(* IEC 61131-3 sources: xpxp/gpt-5, 22 files *)

(* ---- 11.st ---- *)
FUNCTION Sign : INT
VAR_INPUT
    x : REAL;
END_VAR
IF x > 0.0 THEN
    Sign := 1;
ELSIF x < 0.0 THEN
    Sign := -1;
ELSE
    Sign := 0;
END_IF;
RETURN;
END_FUNCTION

(* ---- 14.st ---- *)
FUNCTION FC1001 : BOOL
VAR_INPUT
	MEW: REAL; // Measured value
	SP: REAL;  // Switching value (setpoint)
	HYS: REAL; // Hysteresis in percent of |SP|
END_VAR
VAR_IN_OUT
 	OUT:BOOL;  // Latched output state
END_VAR
VAR
 	P_HYS: REAL; // Absolute hysteresis value derived from percent
END_VAR

// Calculate absolute hysteresis; ensure non-negative percentage
IF HYS < 0.0 THEN
	P_HYS := 0.0;
ELSE
	P_HYS := ABS(SP) * HYS * 0.01;
END_IF

// Hysteresis behavior:
// - Turn ON when measured value exceeds SP
// - Turn OFF when measured value falls below SP - P_HYS
// - Otherwise, retain previous state to avoid fluttering
IF MEW > SP THEN
	OUT := TRUE;
ELSIF MEW < (SP - P_HYS) THEN
	OUT := FALSE;
END_IF

// Function result mirrors the output state
FC1001 := OUT;
RETURN;

(* ---- 15.st ---- *)
FUNCTION FC1002 : BOOL
VAR_INPUT
	E_A, SENSOR: BOOL;
	ZEITW: TIME;
END_VAR
VAR_IN_OUT
	ZEIT:TON;
	P_HU, P_AL: BOOL;
END_VAR

(* Drive timer based on system enable and sensor *)
ZEIT(IN := (E_A AND SENSOR), PT := ZEITW);

(* Alarm latch logic *)
IF NOT E_A THEN
	P_AL := FALSE;
ELSE
	IF P_AL THEN
		P_AL := TRUE; (* keep latched until system is turned off *)
	ELSIF ZEIT.Q THEN
		P_AL := TRUE; (* latch alarm after sustained detection *)
	ELSE
		P_AL := FALSE;
	END_IF
END_IF

(* Horn logic: active only during early detection window *)
IF E_A THEN
	IF SENSOR AND NOT P_AL THEN
		P_HU := TRUE;
	ELSE
		P_HU := FALSE;
	END_IF
ELSE
	P_HU := FALSE;
END_IF

(* Function return indicates system ON status *)
FC1002 := E_A;

(* ---- 18.st ---- *)
FUNCTION FC1003 : VOID
VAR_INPUT
    IN_R:REAL;
    IN_MAX, IN_MIN:REAL;
    OUT_MAX, OUT_MIN:REAL;
END_VAR
VAR_OUTPUT
    OUT_R:REAL;
    FEH:BOOL;
END_VAR
VAR_TEMP
    DIFF1, DIFF2:REAL;
END_VAR

(* Initialize error flag *)
FEH := FALSE;

(* Calculate input and output spans *)
DIFF1 := IN_MAX - IN_MIN;
DIFF2 := OUT_MAX - OUT_MIN;

(* Validate input span to avoid division by zero *)
IF ABS(DIFF1) <= 1.0e-30 THEN
    FEH := TRUE;
    OUT_R := OUT_MIN; (* Safe fallback output *)
    RETURN;
END_IF

(* Normalize input to 0..1 with saturation *)
OUT_R := (IN_R - IN_MIN) / DIFF1;
IF OUT_R < 0.0 THEN
    OUT_R := 0.0;
ELSIF OUT_R > 1.0 THEN
    OUT_R := 1.0;
END_IF

(* Scale to output range *)
OUT_R := OUT_MIN + OUT_R * DIFF2;

END_FUNCTION

(* ---- 1.st ---- *)
FUNCTION_BLOCK FB_AlarmManager
VAR
	xAllOn : BOOL;
	xAllOff : BOOL;

	xAlarm1 : BOOL;
    xAlarm2 : BOOL;
END_VAR

IF xAllOff THEN
	xAlarm1 := FALSE;
	xAlarm2 := FALSE;
	xAllOff := FALSE;
	xAllOn := FALSE;
ELSIF xAllOn THEN
	xAlarm1 := TRUE;
	xAlarm2 := TRUE;
	xAllOn := FALSE;
END_IF

END_FUNCTION_BLOCK

(* ---- 10.st ---- *)
FUNCTION_BLOCK FB_Sigmoid
VAR_INPUT
    X : REAL;
END_VAR
VAR_OUTPUT
    Y : REAL;
END_VAR
VAR
    z : LREAL;    // Intermediate exponential value
    t : LREAL;    // Temporary result in LREAL for precision
END_VAR

// Numerically stable sigmoid implementation:
// if x >= 0: sigmoid(x) = 1 / (1 + exp(-x))
// else:       sigmoid(x) = exp(x) / (1 + exp(x))
IF X >= 0.0 THEN
    z := EXP(LREAL(-X));
    t := 1.0 / (1.0 + z);
    Y := REAL(t);
ELSE
    z := EXP(LREAL(X));
    t := z / (1.0 + z);
    Y := REAL(t);
END_IF
END_FUNCTION_BLOCK

(* ---- 12.st ---- *)
FUNCTION_BLOCK FB_Sinh
VAR
    X : REAL;
END_VAR

(* Compute hyperbolic sine of X in-place using the exponential function.
   Includes simple saturation and piecewise evaluation to mitigate overflow. *)

(* Soft-limit X to a safe computational range for REAL to reduce overflow risk *)
X := LIMIT(-88.0, X, 88.0);

IF X > 80.0 THEN
    (* For large positive X, sinh(X) ≈ 0.5 * exp(X) *)
    X := 0.5 * EXP(X);
ELSIF X < -80.0 THEN
    (* For large negative X, sinh(X) ≈ -0.5 * exp(-X) *)
    X := -0.5 * EXP(-X);
ELSE
    (* General case: sinh(X) = (e^X - e^-X) / 2 *)
    X := 0.5 * (EXP(X) - EXP(-X));
END_IF

END_FUNCTION_BLOCK

(* ---- 13.st ---- *)
FUNCTION_BLOCK FB_FindNumberWithAbort
VAR CONSTANT
    MAXNUMBERS : UINT := 99;
END_VAR
VAR
    aNumbers : ARRAY[0..MAXNUMBERS] OF INT; // Input list of numbers (0..99)
    nCnt : INT;                             // Index/result: 0..99 if found; 100 if not found
END_VAR

// Initialize index
nCnt := 0;

// Search through the list with two abort conditions:
// 1) EXIT when number 10 is found.
// 2) Terminate when end of list is reached (nCnt > MAXNUMBERS).
REPEAT
    IF aNumbers[nCnt] = 10 THEN
        EXIT;
    END_IF
    nCnt := nCnt + 1;
UNTIL nCnt > INT(MAXNUMBERS) END_REPEAT;

(* ---- 16.st ---- *)
FUNCTION_BLOCK FB_TrafficLight
VAR
    North_green : BOOL;
    North_yellow : BOOL;
    North_red : BOOL;
    East_green : BOOL;
    East_yellow : BOOL;
    East_red : BOOL;
    T1 : TON;
END_VAR

(* Free-running 10s cycle using TON *)
T1(IN := NOT T1.Q, PT := T#10s);

(* Default all off *)
North_green := FALSE;
North_yellow := FALSE;
North_red := FALSE;
East_green := FALSE;
East_yellow := FALSE;
East_red := FALSE;

(* Phase selection based on elapsed time *)
IF (T1.ET < T#5s) THEN
    (* 0ms - 5000ms *)
    North_green := TRUE;
    East_red := TRUE;
ELSIF (T1.ET < T#5500ms) THEN
    (* 5000ms - 5500ms *)
    North_yellow := TRUE;
    East_red := TRUE;
ELSIF (T1.ET < T#9500ms) THEN
    (* 5500ms - 9500ms *)
    North_red := TRUE;
    East_green := TRUE;
ELSE
    (* 9500ms - 10000ms *)
    North_red := TRUE;
    East_yellow := TRUE;
END_IF;

END_FUNCTION_BLOCK

(* ---- 17.st ---- *)
FUNCTION_BLOCK FB_WeatherStation
VAR
    aiOutside : INT;       // Outside temperature [°C], read from analog input
    aiHumidity: INT;       // Relative humidity [%]
    sShowText : STRING[80];// Display text for house
END_VAR

// Temperature classification with nested humidity evaluation
IF aiOutside < 18 THEN
    // Below comfort temperature
    sShowText := 'Cold';
ELSIF aiOutside > 25 THEN
    // Above comfort temperature
    sShowText := 'Hot';
ELSE
    // Temperature within 18..25°C: evaluate humidity
    IF (aiHumidity >= 40) AND (aiHumidity <= 75) THEN
        sShowText := 'Opt';
    ELSE
        sShowText := 'Temp. OK';
    END_IF
END_IF

(* ---- 19.st ---- *)
FUNCTION_BLOCK FB1005
VAR_INPUT
    START:BOOL;
    DICKE, V_MAX, V_MIN:REAL;
END_VAR
VAR_OUTPUT
    D_MAX, D_MIN:REAL;
    P1:BOOL;
END_VAR
VAR
    FO:BOOL;
END_VAR

(* Rising edge detection of START: initialize new measurement cycle *)
IF (START AND NOT FO) THEN
    (* Initialize min/max with first sample of the new cycle *)
    D_MAX := DICKE;
    D_MIN := DICKE;
END_IF

(* While measuring, continuously update min/max *)
IF START THEN
    IF DICKE > D_MAX THEN
        D_MAX := DICKE;
    END_IF
    IF DICKE < D_MIN THEN
        D_MIN := DICKE;
    END_IF
END_IF

(* Evaluate reject light based on tolerance band.
   Safety: If V_MIN > V_MAX (invalid band), force reject. *)
IF V_MIN <= V_MAX THEN
    P1 := (D_MIN < V_MIN) OR (D_MAX > V_MAX);
ELSE
    P1 := TRUE;
END_IF

(* Store previous START state for edge detection *)
FO := START
END_FUNCTION_BLOCK

(* ---- 2.st ---- *)
FUNCTION_BLOCK FB_BinomialCoefficient
VAR_INPUT
    N : INT;
    K : INT;
    i : INT;
END_VAR
VAR_OUTPUT
    C : ULINT;
    Valid : BOOL;
    Error : BOOL;
    ErrorID : UINT;
END_VAR
VAR
    nEff : UDINT;
    kEff : UDINT;
    j : UDINT;
    res : ULINT;
    numTerm : ULINT;
    denTerm : ULINT;
    gcd : ULINT;
    temp : ULINT;
    rem : ULINT;
END_VAR

(* Default outputs *)
Error := FALSE;
Valid := FALSE;
ErrorID := UINT#0;
C := ULINT#0;

(* Validate inputs *)
IF (N < 0) OR (K < 0) THEN
    Error := TRUE;
    ErrorID := UINT#10; (* Negative inputs not allowed *)
    RETURN;
END_IF

IF K > N THEN
    Error := TRUE;
    ErrorID := UINT#11; (* K must be <= N *)
    RETURN;
END_IF

(* Prepare effective parameters and use symmetry k = min(K, N-K) *)
nEff := UDINT(N);
kEff := UDINT(K);
IF kEff > (nEff - kEff) THEN
    kEff := nEff - kEff;
END_IF

res := ULINT#1;

(* Trivial cases *)
IF kEff = UDINT#0 THEN
    C := res; (* C(N,0) = 1 *)
    Valid := TRUE;
    RETURN;
END_IF

(* Multiplicative method with GCD reduction to control growth:
   res = product_{j=1..k} (n-k+j)/j
*)
FOR j := UDINT#1 TO kEff DO
    numTerm := ULINT(nEff - kEff + j);  (* numerator term *)
    denTerm := ULINT(j);                 (* denominator term *)

    (* Reduce (res, denTerm) by their GCD *)
    gcd := res;
    temp := denTerm;
    WHILE temp <> ULINT#0 DO
        rem := gcd MOD temp;
        gcd := temp;
        temp := rem;
    END_WHILE
    IF gcd > ULINT#1 THEN
        res := res / gcd;
        denTerm := denTerm / gcd;
    END_IF

    (* Reduce (numTerm, denTerm) by their GCD *)
    gcd := numTerm;
    temp := denTerm;
    WHILE temp <> ULINT#0 DO
        rem := gcd MOD temp;
        gcd := temp;
        temp := rem;
    END_WHILE
    IF gcd > ULINT#1 THEN
        numTerm := numTerm / gcd;
        denTerm := denTerm / gcd;
    END_IF

    (* Apply the reduced multiply/divide step *)
    res := res * numTerm;
    res := res / denTerm;
END_FOR

C := res;
Valid := TRUE
END_FUNCTION_BLOCK

(* ---- 20.st ---- *)
FUNCTION_BLOCK INTERLOCK
VAR_INPUT
    I1 : BOOL;
    I2 : BOOL;
    TL : TIME;
END_VAR
VAR_OUTPUT
    Q1 : BOOL;
    Q2 : BOOL;
END_VAR
VAR
    T1 : TOF;
    T2 : TOF;
END_VAR

(* Clamp the dead time to a minimum of 0 ms *)
IF TL < T#0ms THEN
    T1.PT := T#0ms;
    T2.PT := T#0ms;
ELSE
    T1.PT := TL;
    T2.PT := TL;
END_IF;

(* Timers monitor the opposite output to enforce dead time after switch-off *)
T1.IN := Q2; (* Blocks Q1 while Q2 is TRUE or has been TRUE within TL *)
T2.IN := Q1; (* Blocks Q2 while Q1 is TRUE or has been TRUE within TL *)

(* Execute timers *)
T1();
T2();

(* Interlock logic with deterministic priority to Q1 when both are eligible *)
IF (I1 AND NOT T1.Q) THEN
    Q1 := TRUE;
    Q2 := FALSE;
ELSIF (I2 AND NOT T2.Q) THEN
    Q1 := FALSE;
    Q2 := TRUE;
ELSE
    Q1 := FALSE;
    Q2 := FALSE;
END_IF;

(* ---- 21.st ---- *)
FUNCTION_BLOCK BURNER
VAR_INPUT
    IN : BOOL;
    STAGE2 : BOOL;
    OVER_TEMP : BOOL;
    OIL_TEMP : BOOL := TRUE;
    FLAME : BOOL;
    RST : BOOL;
    RST_TIMER : BOOL;
    PRE_HEAT_TIME : TIME := t#5s;
    PRE_VENT_TIME : TIME := t#15s;
    PRE_IGNITE_TIME : TIME := t#15s;
    POST_IGNITE_TIME : TIME := t#25s;
    STAGE2_DELAY : TIME := t#10s;
    SAFETY_TIME : TIME := t#5s;
    LOCKOUT_TIME : TIME := t#10s;
    MULTIPLE_IGNITION : BOOL := TRUE;
    KW1 : REAL;
    KW2 : REAL;
END_VAR
VAR_OUTPUT
    MOTOR : BOOL;
    COIL1 : BOOL;
    COIL2 : BOOL;
    PRE_HEAT : BOOL;
    IGNITE : BOOL;
    FAIL : BOOL;
    KWH : REAL;
    STATUS : BYTE;
END_VAR
VAR_IN_OUT
    RUNTIME1 : UDINT;
    RUNTIME2 : UDINT;
    CYCLES : UDINT;
END_VAR
VAR
    state : INT;
    last : TIME;
    tx : TIME;
    last_change : TIME;
    timer1 : TON;
    timer2 : TON;
    oil_temp_last : BOOL; (* used as last RST state for rising edge detection *)
    cycles2 : UDINT;      (* snapshot of RUNTIME1 at Stage1 start, used for Stage2 delay *)
END_VAR

(* Initialize to Standby on first scan *)
IF state = 0 THEN
    state := 110; (* Standby *)
    FAIL := FALSE;
    STATUS := 110;
END_IF

(* Reset runtime and energy counters on request *)
IF RST_TIMER THEN
    RUNTIME1 := 0;
    RUNTIME2 := 0;
    CYCLES := 0;
    KWH := 0.0;
    cycles2 := 0;
END_IF

(* Default outputs off; will be enabled per state below *)
MOTOR := FALSE;
COIL1 := FALSE;
COIL2 := FALSE;
PRE_HEAT := FALSE;
IGNITE := FALSE;

(* Over-temperature immediate lockout *)
IF OVER_TEMP AND NOT FAIL THEN
    FAIL := TRUE;
    STATUS := 9; (* boiler overheating contact has tripped *)
    state := 1000; (* Lockout state *)
    (* Prepare lockout timer1 *)
    timer1.IN := TRUE;
    timer1.PT := LOCKOUT_TIME;
END_IF

(* Lockout handling *)
IF state = 1000 THEN
    (* Ensure all actuators are off during lockout *)
    MOTOR := FALSE;
    COIL1 := FALSE;
    COIL2 := FALSE;
    PRE_HEAT := FALSE;
    IGNITE := FALSE;

    (* Run lockout timer *)
    timer1.PT := LOCKOUT_TIME;
    timer1.IN := NOT timer1.Q; (* keep running until elapsed *)

    (* Require RST low during lockout and accept rising edge after timer elapsed *)
    IF timer1.Q THEN
        IF (RST AND NOT oil_temp_last) THEN
            (* Rising edge of RST after lockout time: clear fault and return to standby *)
            FAIL := FALSE;
            state := 110;
            STATUS := 110;
            (* Reset lockout timer *)
            timer1.IN := FALSE;
        END_IF
    END_IF
ELSE
    (* Main sequence state machine when not in lockout *)
    IF state = 110 THEN
        (* Standby *)
        STATUS := 110;
        (* Wait for start command and no over-temp *)
        IF IN AND NOT OVER_TEMP THEN
            (* Start pre-heat phase *)
            state := 111;
            PRE_HEAT := TRUE;
            timer1.IN := TRUE;
            timer1.PT := PRE_HEAT_TIME;
        END_IF

    ELSIF state = 111 THEN
        (* Pre-heat *)
        STATUS := 111;
        PRE_HEAT := TRUE;

        (* Fault if flame detected during pre-heat *)
        IF FLAME THEN
            FAIL := TRUE;
            STATUS := 2;
            state := 1000;
            (* Start lockout timer *)
            timer1.IN := TRUE;
            timer1.PT := LOCKOUT_TIME;
        ELSIF OIL_TEMP THEN
            (* Oil temperature reached: proceed to motor pre-ventilation *)
            PRE_HEAT := FALSE;
            state := 115;
            MOTOR := TRUE;
            (* Determine ignition lead time (clamped to PRE_VENT_TIME) *)
            tx := PRE_IGNITE_TIME;
            IF tx > PRE_VENT_TIME THEN
                tx := PRE_VENT_TIME;
            END_IF
            (* First pre-ventilation interval: until ignition turn-on *)
            timer1.IN := TRUE;
            timer1.PT := PRE_VENT_TIME - tx;
        ELSIF timer1.Q AND (NOT OIL_TEMP) THEN
            (* Pre-heat timeout without oil temp *)
            FAIL := TRUE;
            STATUS := 1;
            state := 1000;
            (* Start lockout timer *)
            timer1.IN := TRUE;
            timer1.PT := LOCKOUT_TIME;
        END_IF

    ELSIF state = 115 THEN
        (* Pre-ventilation part 1: fan only until ignition turn-on *)
        STATUS := 111;
        MOTOR := TRUE;
        (* Fault if flame during aeration *)
        IF FLAME THEN
            FAIL := TRUE;
            STATUS := 3;
            state := 1000;
            timer1.IN := TRUE;
            timer1.PT := LOCKOUT_TIME;
        ELSIF timer1.Q THEN
            (* Turn on ignition and wait remaining time to open valve *)
            state := 116;
            MOTOR := TRUE;
            IGNITE := TRUE;
            (* tx holds the ignition lead time *)
            timer1.IN := TRUE;
            timer1.PT := tx;
        END_IF

    ELSIF state = 116 THEN
        (* Pre-ventilation part 2: ignition running, waiting to open valve *)
        STATUS := 111;
        MOTOR := TRUE;
        IGNITE := TRUE;
        (* Fault if flame during aeration *)
        IF FLAME THEN
            FAIL := TRUE;
            STATUS := 3;
            state := 1000;
            timer1.IN := TRUE;
            timer1.PT := LOCKOUT_TIME;
        ELSIF timer1.Q THEN
            (* Open oil valve and start safety timer *)
            state := 130;
            MOTOR := TRUE;
            COIL1 := TRUE;
            IGNITE := TRUE;
            timer1.IN := TRUE;
            timer1.PT := SAFETY_TIME;
        END_IF

    ELSIF state = 130 THEN
        (* Oil valve open, safety time for flame establishment *)
        STATUS := 111;
        MOTOR := TRUE;
        COIL1 := TRUE;
        IGNITE := TRUE;

        IF FLAME THEN
            (* Successful flame: go to Stage 1 run *)
            state := 112;
            CYCLES := CYCLES + 1;
            cycles2 := RUNTIME1; (* snapshot for Stage2 delay *)
            (* Begin post-ignition hold *)
            timer1.IN := TRUE;
            timer1.PT := POST_IGNITE_TIME;
        ELSIF timer1.Q THEN
            (* Safety time expired without flame *)
            FAIL := TRUE;
            STATUS := 4;
            state := 1000;
            timer1.IN := TRUE;
            timer1.PT := LOCKOUT_TIME;
        END_IF

    ELSIF state = 112 THEN
        (* Burner runs on Stage 1 *)
        STATUS := 112;
        MOTOR := TRUE;
        COIL1 := TRUE;
        (* Post-ignition handling *)
        IF NOT timer1.Q THEN
            IGNITE := TRUE;
        ELSE
            IGNITE := FALSE;
            timer1.IN := FALSE; (* stop post-ignition timer once complete *)
        END_IF

        (* Stage 2 auto activation after delay when requested *)
        IF STAGE2 THEN
            IF (RUNTIME1 >= cycles2 + (TIME_TO_UDINT(STAGE2_DELAY) / 1000)) THEN
                state := 113;
                (* keep IGNITE as per post-ignition timer state *)
            END_IF
        END_IF

        (* Flame loss handling *)
        IF NOT FLAME THEN
            IF MULTIPLE_IGNITION THEN
                state := 160; (* Re-ignition Stage 1 *)
                IGNITE := TRUE;
                timer1.IN := TRUE;
                timer1.PT := SAFETY_TIME;
            ELSE
                FAIL := TRUE;
                STATUS := 5;
                state := 1000;
                timer1.IN := TRUE;
                timer1.PT := LOCKOUT_TIME;
            END_IF
        END_IF

    ELSIF state = 113 THEN
        (* Burner runs on Stage 2 *)
        STATUS := 113;
        MOTOR := TRUE;
        COIL1 := TRUE;
        COIL2 := TRUE;
        (* Post-ignition handling continues if active *)
        IF NOT timer1.Q THEN
            IGNITE := TRUE;
        ELSE
            IGNITE := FALSE;
            timer1.IN := FALSE;
        END_IF

        (* Allow dropping back to Stage 1 if STAGE2 request is removed *)
        IF NOT STAGE2 THEN
            state := 112;
        END_IF

        (* Flame loss handling *)
        IF NOT FLAME THEN
            IF MULTIPLE_IGNITION THEN
                state := 161; (* Re-ignition Stage 2 *)
                IGNITE := TRUE;
                timer1.IN := TRUE;
                timer1.PT := SAFETY_TIME;
            ELSE
                FAIL := TRUE;
                STATUS := 5;
                state := 1000;
                timer1.IN := TRUE;
                timer1.PT := LOCKOUT_TIME;
            END_IF
        END_IF

    ELSIF state = 160 THEN
        (* Re-ignition attempt on Stage 1 *)
        STATUS := 112;
        MOTOR := TRUE;
        COIL1 := TRUE;
        IGNITE := TRUE;
        IF FLAME THEN
            (* Flame re-established: continue run with post-ignition *)
            state := 112;
            timer1.IN := TRUE;
            timer1.PT := POST_IGNITE_TIME;
        ELSIF timer1.Q THEN
            (* Re-ignition failed *)
            FAIL := TRUE;
            STATUS := 5;
            state := 1000;
            timer1.IN := TRUE;
            timer1.PT := LOCKOUT_TIME;
        END_IF

    ELSIF state = 161 THEN
        (* Re-ignition attempt on Stage 2 *)
        STATUS := 113;
        MOTOR := TRUE;
        COIL1 := TRUE;
        COIL2 := TRUE;
        IGNITE := TRUE;
        IF FLAME THEN
            (* Flame re-established: continue run with post-ignition *)
            state := 113;
            timer1.IN := TRUE;
            timer1.PT := POST_IGNITE_TIME;
        ELSIF timer1.Q THEN
            (* Re-ignition failed *)
            FAIL := TRUE;
            STATUS := 5;
            state := 1000;
            timer1.IN := TRUE;
            timer1.PT := LOCKOUT_TIME;
        END_IF
    END_IF
END_IF

(* Second counter and energy metering *)
(* Generate 1-second tick while burner is in either stage or during re-ignition attempts *)
timer2.PT := T#1s;
IF (state = 112) OR (state = 113) OR (state = 160) OR (state = 161) THEN
    timer2.IN := NOT timer2.Q;
ELSE
    timer2.IN := FALSE;
END_IF

(* Execute timers *)
timer1();
timer2();

(* On 1-second tick, accumulate runtimes and energy *)
IF timer2.Q THEN
    IF (state = 112) OR (state = 160) THEN
        RUNTIME1 := RUNTIME1 + 1;
        KWH := KWH + (KW1 / 3600.0);
    ELSIF (state = 113) OR (state = 161) THEN
        RUNTIME2 := RUNTIME2 + 1;
        KWH := KWH + (KW2 / 3600.0);
    END_IF
END_IF

(* Update previous RST state for rising edge detection *)
oil_temp_last := RST;

(* ---- 22.st ---- *)
FUNCTION_BLOCK FB_ArmHomeWorkController
VAR_INPUT
    MoveToWorkCmd    : BOOL; // Momentary command to move towards Work position
    MoveToHomeCmd    : BOOL; // Momentary command to move towards Home position
    AtWorkSensor     : BOOL; // TRUE only when arm is exactly at Work position
    AtHomeSensor     : BOOL; // TRUE only when arm is exactly at Home position
    MovementPermitted: BOOL; // Global safety interlock; movement allowed only if TRUE
END_VAR
VAR_OUTPUT
    MotorForward : BOOL; // Energize motor towards Work
    MotorReverse : BOOL; // Energize motor towards Home
END_VAR
VAR
    prevMoveToWorkCmd : BOOL; // Previous state for rising edge detection
    prevMoveToHomeCmd : BOOL; // Previous state for rising edge detection
    riseWork          : BOOL; // Rising edge of MoveToWorkCmd
    riseHome          : BOOL; // Rising edge of MoveToHomeCmd
    forwardLatched    : BOOL; // Latched request to move forward (to Work)
    reverseLatched    : BOOL; // Latched request to move reverse (to Home)
END_VAR

// Rising edge detection for commands
riseWork := MoveToWorkCmd AND NOT prevMoveToWorkCmd;
riseHome := MoveToHomeCmd AND NOT prevMoveToHomeCmd;

// Safety interlock handling and core sequencing
IF NOT MovementPermitted THEN
    // Immediate stop and require new command after safety returns
    forwardLatched := FALSE;
    reverseLatched := FALSE;
ELSE
    // Auto-stop when target position sensor becomes TRUE
    IF AtWorkSensor THEN
        forwardLatched := FALSE;
    END_IF;
    IF AtHomeSensor THEN
        reverseLatched := FALSE;
    END_IF;

    // Process new commands (momentary). Opposite direction is canceled.
    // If both commands occur simultaneously, Home has priority (processed last).
    IF riseWork AND NOT AtWorkSensor THEN
        forwardLatched := TRUE;
        reverseLatched := FALSE;
    END_IF;

    IF riseHome AND NOT AtHomeSensor THEN
        reverseLatched := TRUE;
        forwardLatched := FALSE;
    END_IF;
END_IF;

// Output interlocks: Never allow both directions active, and do not drive if already at target
MotorForward := MovementPermitted AND forwardLatched AND NOT AtWorkSensor AND NOT reverseLatched;
MotorReverse := MovementPermitted AND reverseLatched AND NOT AtHomeSensor AND NOT forwardLatched;

// Update previous states for edge detection
prevMoveToWorkCmd := MoveToWorkCmd;
prevMoveToHomeCmd := MoveToHomeCmd;
END_FUNCTION_BLOCK

(* ---- 3.st ---- *)
FUNCTION_BLOCK FB_Fibonacci
VAR_INPUT
    X : INT;
END_VAR
VAR
    t1 : DINT; // Current Fibonacci number F(n)
    t2 : DINT; // Helper holding F(n+1) during iteration
    x_tmp : INT; // Clamped copy of X used as loop counter
END_VAR

// Clamp input to safe range to avoid DINT overflow (F(46) fits in 32-bit signed)
IF X < 0 THEN
    x_tmp := 0;
ELSIF X > 46 THEN
    x_tmp := 46;
ELSE
    x_tmp := X;
END_IF

// Initialize base values: F(0) = 0, F(1) = 1
t1 := 0;
t2 := 1;

// Iteratively compute Fibonacci using in-place update without extra temp variable
WHILE x_tmp > 0 DO
    t2 := t1 + t2;   // t2 becomes F(n) + F(n+1) = F(n+2)
    t1 := t2 - t1;   // t1 becomes previous t2 = F(n+1)
    x_tmp := x_tmp - 1;
END_WHILE
END_FUNCTION_BLOCK

(* ---- 4.st ---- *)
FUNCTION_BLOCK FB_FillLevelCheck
VAR
    aiLevel : INT;
    PercentLevel : UINT;
    doLow : BOOL;
    doOk : BOOL;
    doHigh : BOOL;
    doAlarm : BOOL;
END_VAR

(* Scale raw input (0..32767) to 0..100% with clamping *)
IF aiLevel <= 0 THEN
    PercentLevel := 0;
ELSIF aiLevel >= 32767 THEN
    PercentLevel := 100;
ELSE
    PercentLevel := UINT((UDINT(aiLevel) * UDINT(100)) / UDINT(32767));
END_IF
END_IF

(* Alarm if below 1% *)
doAlarm := (PercentLevel < 1);

(* Default outputs *)
doLow := FALSE;
doOk := FALSE;
doHigh := FALSE;

(* Range classification using CASE *)
CASE PercentLevel OF
    0..20:
        doLow := TRUE;
    21..80:
        doOk := TRUE;
    81..100:
        doHigh := TRUE;
ELSE
    (* Should not occur due to clamping above *)
END_CASE
END_FUNCTION_BLOCK

(* ---- 5.st ---- *)
FUNCTION_BLOCK FB_GateController
VAR
    Start_Loop : BOOL := FALSE;
    one_hour : TIME := T#1h;
    One_Hour_Timer : TON;
    Gate_Open : BOOL := FALSE;
    Close_Gate_Inst : BOOL := FALSE;
    Sensed_Car : BOOL := FALSE;
    Sensed_Car_Inst : BOOL := FALSE;
    Sensed_App : BOOL := FALSE;
    Mobile_Inst : BOOL := FALSE;
    Auth : STRING;
    my_defined_str : STRING := 'abcd';
END_VAR

(* Start the one-hour timer when Start_Loop is FALSE *)
One_Hour_Timer(IN := NOT Start_Loop, PT := one_hour);

(* Open gate on valid authorization and presence of app or car *)
IF (Auth = my_defined_str) THEN
    IF (Sensed_App OR Sensed_Car) THEN
        Gate_Open := TRUE;
    END_IF
END_IF

(* Close gate on timer timeout (use Sensed_Car_Inst as previous Q memory for rising edge) *)
IF (One_Hour_Timer.Q AND NOT Sensed_Car_Inst) THEN
    IF Gate_Open THEN
        Close_Gate_Inst := TRUE;
        Gate_Open := FALSE;
    ELSE
        Close_Gate_Inst := FALSE;
    END_IF
    Sensed_Car_Inst := TRUE;
ELSE
    Close_Gate_Inst := FALSE;
    IF NOT One_Hour_Timer.Q THEN
        Sensed_Car_Inst := FALSE;
    END_IF
END_IF

(* ---- 6.st ---- *)
FUNCTION_BLOCK FB_CraneLift
VAR CONSTANT
    WAIT : UINT:= 0;
    TOP_POSITION : UINT:= 1;
    BOTTOM_POSITION : UINT:= 2;
    GETBOX : UINT:= 3;
    UNLOAD_POSITION : UINT:= 4;
    UNLOAD_BOX : UINT:= 5;
END_VAR

VAR
    (*-- digital outputs*)
    doConvTop: BOOL;
    doConvBottom: BOOL;
    doConvLift: BOOL;
    doLiftTop: BOOL;
    doLiftBottom: BOOL;
    doLiftUnload: BOOL;
    (*-- digital inputs*)
    diConvTop: BOOL;
    diConvBottom: BOOL;
    diLiftTop: BOOL;
    diLiftBottom: BOOL;
    diLiftUnload: BOOL;
    diBoxLift: BOOL;
    (*-- status variables*)
    selectLift: UINT;
    ConvTopOn: BOOL;
    ConvBottomOn: BOOL;
END_VAR

(* Default outputs to safe state *)
doLiftTop := FALSE;
doLiftBottom := FALSE;
doLiftUnload := FALSE;
doConvLift := FALSE;

(* Source conveyors: run while light barrier is free *)
ConvTopOn := NOT diConvTop;
ConvBottomOn := NOT diConvBottom;
doConvTop := ConvTopOn;
doConvBottom := ConvBottomOn;

(* State machine *)
IF selectLift = WAIT THEN
    (* Request lift based on waiting crate(s); priority: top then bottom *)
    IF diConvTop THEN
        selectLift := TOP_POSITION;
    ELSIF diConvBottom THEN
        selectLift := BOTTOM_POSITION;
    END_IF

ELSIF selectLift = TOP_POSITION THEN
    IF diLiftTop THEN
        selectLift := GETBOX;
    ELSE
        doLiftTop := TRUE;
    END_IF

ELSIF selectLift = BOTTOM_POSITION THEN
    IF diLiftBottom THEN
        selectLift := GETBOX;
    ELSE
        doLiftBottom := TRUE;
    END_IF

ELSIF selectLift = GETBOX THEN
    (* Pull crate onto lift until fully on the lift *)
    IF diBoxLift THEN
        doConvLift := FALSE;
        selectLift := UNLOAD_POSITION;
    ELSE
        doConvLift := TRUE;
    END_IF

ELSIF selectLift = UNLOAD_POSITION THEN
    IF diLiftUnload THEN
        selectLift := UNLOAD_BOX;
    ELSE
        doLiftUnload := TRUE;
    END_IF

ELSIF selectLift = UNLOAD_BOX THEN
    (* Convey crate off the lift until it has left *)
    IF NOT diBoxLift THEN
        doConvLift := FALSE;
        selectLift := WAIT;
    ELSE
        doConvLift := TRUE;
    END_IF

ELSE
    (* Fallback to safe idle *)
    selectLift := WAIT;
END_IF
END_FUNCTION_BLOCK

(* ---- 7.st ---- *)
FUNCTION_BLOCK FB_CraneLoad
VAR CONSTANT
    MAX_INDEX: USINT := 4; // Highest index (0..4 -> 5 load receptors)
END_VAR
VAR
    aWeights : ARRAY[0..MAX_INDEX] OF INT; // Analog inputs 0..32767
    iCnt : USINT;                          // Loop counter
    sumWeight : DINT;                      // Total load (use DINT to avoid overflow)
    avgWeight : INT;                       // Average load per receptor
END_VAR

// Reset sum each cycle
sumWeight := DINT#0;

// Sum all load receptor values using FOR loop
FOR iCnt := USINT#0 TO MAX_INDEX DO
    sumWeight := sumWeight + DINT(aWeights[iCnt]);
END_FOR

// Compute average: total divided by number of receptors (MAX_INDEX + 1)
avgWeight := INT(sumWeight / (DINT(MAX_INDEX) + DINT#1));

END_FUNCTION_BLOCK

(* ---- 8.st ---- *)
FUNCTION_BLOCK FB_LambertW
VAR_INPUT
    X : REAL;
END_VAR
VAR
    w : REAL;
    i : INT;
    we : REAL;
    w1e : REAL;
    ewx : REAL;
    last : DWORD;
END_VAR

(* Handle domain boundary and initial guess *)
ewx := -EXP(-1.0);
IF X <= ewx THEN
    (* At or below the branch point, return -1 on principal branch *)
    w := -1.0;
ELSE
    (* Initial guess selection *)
    IF X < -0.3 THEN
        (* Near the branch point use a square-root based approximation *)
        we := EXP(1.0) * X + 1.0;
        IF we > 0.0 THEN
            w := -1.0 + SQRT(2.0 * we);
        ELSE
            w := -0.5;
        END_IF
    ELSIF X < 3.0 THEN
        (* Moderate values: log1p approximation *)
        w := LN(1.0 + X);
    ELSE
        (* Large values: asymptotic expansion *)
        w := LN(X) - LN(LN(X));
    END_IF

    (* Halley's method iterations *)
    FOR i := 0 TO 19 DO
        (* f = w*exp(w) - x *)
        ewx := EXP(w);
        we := w * ewx;
        w1e := we - X;

        (* denom = exp(w)*(w+1) - (w+2)*f/(2*(w+1)) *)
        ewx := (ewx * (w + 1.0)) - ((w + 2.0) * w1e) / (2.0 * (w + 1.0));

        (* Update: w := w - f/denom *)
        w1e := w1e / ewx;
        w := w - w1e;

        (* Convergence check *)
        IF ABS(w1e) <= 1.0E-6 * (1.0 + ABS(w)) THEN
            EXIT;
        END_IF
    END_FOR
END_IF
END_FUNCTION_BLOCK

(* ---- 9.st ---- *)
FUNCTION_BLOCK FB_LeapYearCheck
VAR_INPUT
    YEAR : INT;
END_VAR
VAR_OUTPUT
    IsLeapYear : BOOL;
END_VAR

IF YEAR > 0 THEN
    IF YEAR MOD 4 = 0 THEN
        IF YEAR MOD 100 = 0 THEN
            IF YEAR MOD 400 = 0 THEN
                IsLeapYear := TRUE;
            ELSE
                IsLeapYear := FALSE;
            END_IF
        ELSE
            IsLeapYear := TRUE;
        END_IF
    ELSE
        IsLeapYear := FALSE;
    END_IF
ELSE
    IsLeapYear := FALSE;
END_IF
